// Numeric helper namespace.
PROGRAM Math
VAR
END_VAR

// Time-compensated smoothing coefficient clamped to 0..1.
METHOD ExptDecay : LREAL
VAR_INPUT
    rBlendFactor : LREAL;   // Base blend factor, clamped 0..1.
    rDeltaTime   : LREAL := 0.01;   // Sample time in seconds.
END_VAR
rBlendFactor := LIMIT(0.0, rBlendFactor, 1.0);
rDeltaTime   := MAX(rDeltaTime, 0.0);
ExptDecay := LIMIT(0.0, 1.0 - EXPT(1.0 - rBlendFactor, rDeltaTime), 1.0);
END_METHOD

// Low-pass coefficient from cutoff frequency; clamped to 0..1.
METHOD FreqCutoffCoef : LREAL
VAR_STAT CONSTANT
	rA: LREAL := 2.0 * 3.141592653589793;
END_VAR
VAR_INPUT
    rCutoffHz  : LREAL;   // Cutoff frequency in Hz.
    rDeltaTime : LREAL;   // Sample time in seconds.
END_VAR
VAR
	rOmega : LREAL;
END_VAR
rCutoffHz  := MAX(rCutoffHz, 0.0);
rDeltaTime := MAX(rDeltaTime, 0.0);
rOmega := rA * rCutoffHz;
FreqCutoffCoef := 1.0 - EXP(-rOmega * rDeltaTime);
FreqCutoffCoef := LIMIT(0.0, FreqCutoffCoef, 1.0);
END_METHOD

// Scales rX from input range to output range; returns 0 when input span is 0.
METHOD LinearScale : LREAL
VAR_INPUT
	rX				: LREAL; // Input value.
	rMinX			: LREAL; // Input range minimum.
	rMaxX			: LREAL; // Input range maximum.
	rMinY			: LREAL := 0; // Output range minimum.
	rMaxY			: LREAL := 1; // Output range maximum.
END_VAR
VAR
	_rDnmtr			: LREAL := rMaxX - rMinX;
END_VAR
IF _rDnmtr <> 0 THEN
	LinearScale := rMinY + ((rX - rMinX)/_rDnmtr) * (rMaxY - rMinY);
END_IF
END_METHOD

// First-order filter output.
METHOD LowPassFilter : LREAL
VAR_INPUT
	rX				: LREAL; // New input.
	rPrvY			: LREAL; // Previous output.
	
	rCoefficient	: LREAL; // Blend coefficient, normally 0..1.
END_VAR
LowPassFilter := rX * rCoefficient + rPrvY * (1 - rCoefficient);
END_METHOD

// Returns pseudo-random LREAL.
METHOD Random : LREAL
VAR_STAT
	_nSeed		: INT;
END_VAR
VAR
	_drand		: Tc2_System.DRAND;
END_VAR
_drand(Seed := _nSeed, Num => Random);
_nSeed := _nSeed + 1;
END_METHOD

// Rounds rValue at decimal position nPosition.
METHOD Round : LREAL
VAR_INPUT
	rValue: LREAL; // Value to round.
	nPosition: SINT; // Decimal position.
END_VAR
VAR
	rFactor: LREAL := 0;
	rTemp: LINT := 0;
END_VAR
rFactor := EXPT(10, -nPosition);
rTemp := LREAL_TO_LINT(rValue * rFactor);
Round := LINT_TO_LREAL(rTemp) / rFactor;
END_METHOD

END_PROGRAM

(* stored: Version 1.1.0.1
   POU Math: Id {79849915-ccca-45cc-a51a-353bb7315daa}, SpecialFunc None
   Method ExptDecay: Id {8d3aa407-7a4a-435a-88e6-4592a7a47b65}
   Method FreqCutoffCoef: Id {bd72f08d-8d4f-43e5-b950-5b0461356dd2}
   Method LinearScale: Id {57ad8d01-8b3d-4c66-a03e-ccd8286efe23}
   Method LowPassFilter: Id {8bf1a163-e19a-406a-9e5d-a23ea6bfa2ad}
   Method Random: Id {446e7349-8d3a-44ca-b827-be8536ff03cb}
   Method Round: Id {34e0d5ed-7b8b-4a67-875b-cea49a04c3c3} *)
